// TIA Portal project "Trapano" (V15.1)

(* hardware
DEVICE "S7-1200 station_1"  S7-1200 Station
   slot 0: "Telaio di montaggio_0"  S7-1200 Rack  Rack  V1.0
   slot 1: "PLC_1"  CPU 1214C DC/DC/DC  6ES7 214-1AG40-0XB0  V4.2
*)

// ===== PLC "PLC_1"  CPU 1214C DC/DC/DC =====

VAR_GLOBAL   // PLC tag table "Tabella delle variabili standard"
   "y" AT %I0.0 : Bool;
   "x" AT %I0.1 : Bool;
   "a" AT %I0.2 : Bool;
   "b" AT %I0.3 : Bool;
   "start" AT %I0.4 : Bool;
   "m" AT %I0.5 : Bool;
   "down" AT %Q0.0 : Bool;
   "up" AT %Q0.1 : Bool;
   "rotate" AT %Q0.2 : Bool;
   "oil" AT %Q0.3 : Bool;
END_VAR

VAR_GLOBAL CONSTANT   // PLC tag table "Tabella delle variabili standard"
   "tempo_raffreddamento" : Time := T#5s;
END_VAR

DATA_BLOCK "variabili_stato"   // DB1
{ S7_Optimized_Access := 'TRUE' }
VERSION : 0.1
   VAR RETAIN
      home : Bool := true;
      scendi : Bool;
      pezzo_alto : Bool;
      pezzo_alto_risalita : Bool;
      lubrifica : Bool;
      foro : Bool;
      sali : Bool;
      wait : Bool;
   END_VAR
BEGIN
END_DATA_BLOCK

// folder: System blocks/Program resources

DATA_BLOCK "IEC_Timer_0_DB"   // DB2
{ S7_Optimized_Access := 'TRUE' }
AUTHOR : Simatic
FAMILY : IEC
NAME : IEC_TMR
VERSION : 1.0
// stored: InstanceOfName IEC_TIMER
"IEC_TIMER"
BEGIN
END_DATA_BLOCK

// folder: (top level)

ORGANIZATION_BLOCK "Main"   // OB1, LAD, ProgramCycle
TITLE = "Main Program Sweep (Cycle)"
{ S7_Optimized_Access := 'TRUE' }
VERSION : 0.1
   VAR_INPUT
      Initial_Call : Bool;   // Initial call of this OB
      Remanence : Bool;   // =True, if remanent data are available
   END_VAR
   VAR_TEMP   // added for the SCL form of the ladder/FBD networks
      _w1 : Bool;
   END_VAR
BEGIN

REGION Network 1
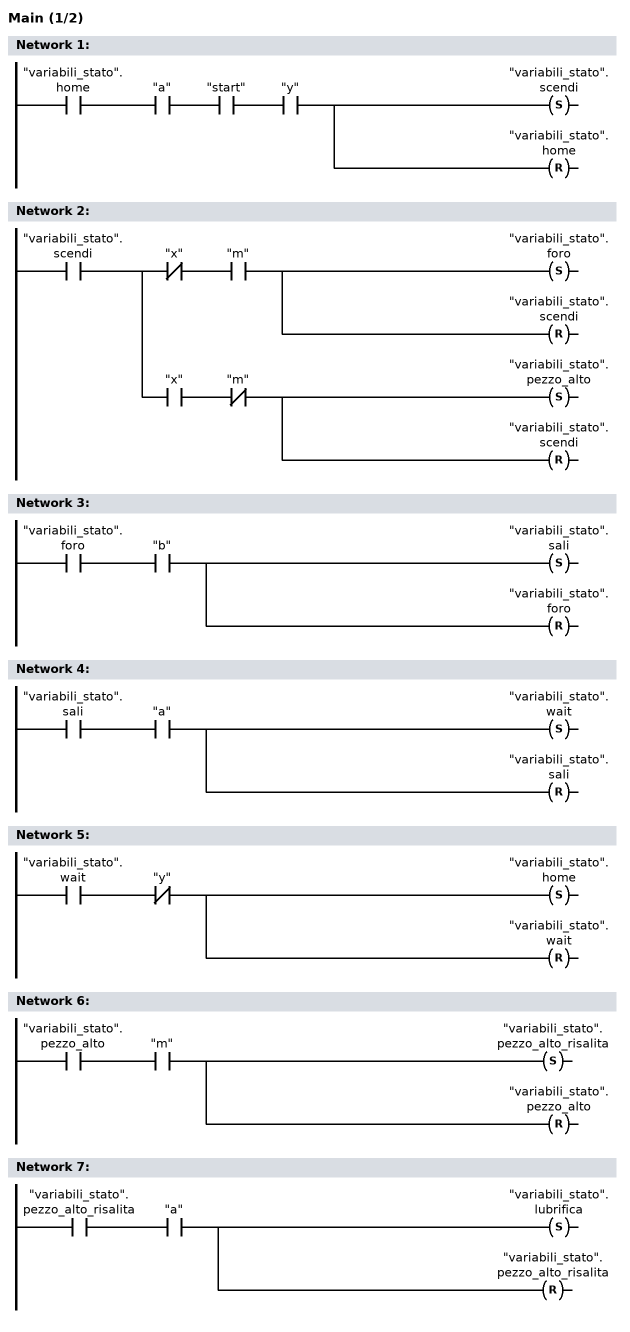
   RUNG wire#powerrail
      Contact( "variabili_stato".home )
      Contact( "a" )
      Contact( "start" )
      Contact( "y" )
      wire#w1
      S_Coil( "variabili_stato".scendi )
   END_RUNG
   RUNG wire#w1
      R_Coil( "variabili_stato".home )
   END_RUNG
   // the same network as SCL:
   IF "variabili_stato".home AND "a" AND "start" AND "y" THEN
       "variabili_stato".scendi := TRUE;
       "variabili_stato".home := FALSE;
   END_IF;
END_REGION

REGION Network 2
   RUNG wire#powerrail
      Contact( "variabili_stato".scendi )
      wire#w1
      I_Contact( "x" )
      Contact( "m" )
      wire#w2
      S_Coil( "variabili_stato".foro )
   END_RUNG
   RUNG wire#w2
      R_Coil( "variabili_stato".scendi )
   END_RUNG
   RUNG wire#w1
      Contact( "x" )
      I_Contact( "m" )
      wire#w3
      S_Coil( "variabili_stato".pezzo_alto )
   END_RUNG
   RUNG wire#w3
      R_Coil( "variabili_stato".scendi )
   END_RUNG
   // the same network as SCL:
   IF "variabili_stato".scendi AND NOT "x" AND "m" THEN "variabili_stato".foro := TRUE; END_IF;
   #_w1 := "variabili_stato".scendi;
   IF "variabili_stato".scendi AND NOT "x" AND "m" THEN "variabili_stato".scendi := FALSE; END_IF;
   IF #_w1 AND "x" AND NOT "m" THEN
       "variabili_stato".pezzo_alto := TRUE;
       "variabili_stato".scendi := FALSE;
   END_IF;
END_REGION

REGION Network 3
   RUNG wire#powerrail
      Contact( "variabili_stato".foro )
      Contact( "b" )
      wire#w1
      S_Coil( "variabili_stato".sali )
   END_RUNG
   RUNG wire#w1
      R_Coil( "variabili_stato".foro )
   END_RUNG
   // the same network as SCL:
   IF "variabili_stato".foro AND "b" THEN
       "variabili_stato".sali := TRUE;
       "variabili_stato".foro := FALSE;
   END_IF;
END_REGION

REGION Network 4
   RUNG wire#powerrail
      Contact( "variabili_stato".sali )
      Contact( "a" )
      wire#w1
      S_Coil( "variabili_stato".wait )
   END_RUNG
   RUNG wire#w1
      R_Coil( "variabili_stato".sali )
   END_RUNG
   // the same network as SCL:
   IF "variabili_stato".sali AND "a" THEN
       "variabili_stato".wait := TRUE;
       "variabili_stato".sali := FALSE;
   END_IF;
END_REGION

REGION Network 5
   RUNG wire#powerrail
      Contact( "variabili_stato".wait )
      I_Contact( "y" )
      wire#w1
      S_Coil( "variabili_stato".home )
   END_RUNG
   RUNG wire#w1
      R_Coil( "variabili_stato".wait )
   END_RUNG
   // the same network as SCL:
   IF "variabili_stato".wait AND NOT "y" THEN
       "variabili_stato".home := TRUE;
       "variabili_stato".wait := FALSE;
   END_IF;
END_REGION

REGION Network 6
   RUNG wire#powerrail
      Contact( "variabili_stato".pezzo_alto )
      Contact( "m" )
      wire#w1
      S_Coil( "variabili_stato".pezzo_alto_risalita )
   END_RUNG
   RUNG wire#w1
      R_Coil( "variabili_stato".pezzo_alto )
   END_RUNG
   // the same network as SCL:
   IF "variabili_stato".pezzo_alto AND "m" THEN
       "variabili_stato".pezzo_alto_risalita := TRUE;
       "variabili_stato".pezzo_alto := FALSE;
   END_IF;
END_REGION

REGION Network 7
   RUNG wire#powerrail
      Contact( "variabili_stato".pezzo_alto_risalita )
      Contact( "a" )
      wire#w1
      S_Coil( "variabili_stato".lubrifica )
   END_RUNG
   RUNG wire#w1
      R_Coil( "variabili_stato".pezzo_alto_risalita )
   END_RUNG
   // the same network as SCL:
   IF "variabili_stato".pezzo_alto_risalita AND "a" THEN
       "variabili_stato".lubrifica := TRUE;
       "variabili_stato".pezzo_alto_risalita := FALSE;
   END_IF;
END_REGION

REGION Network 8
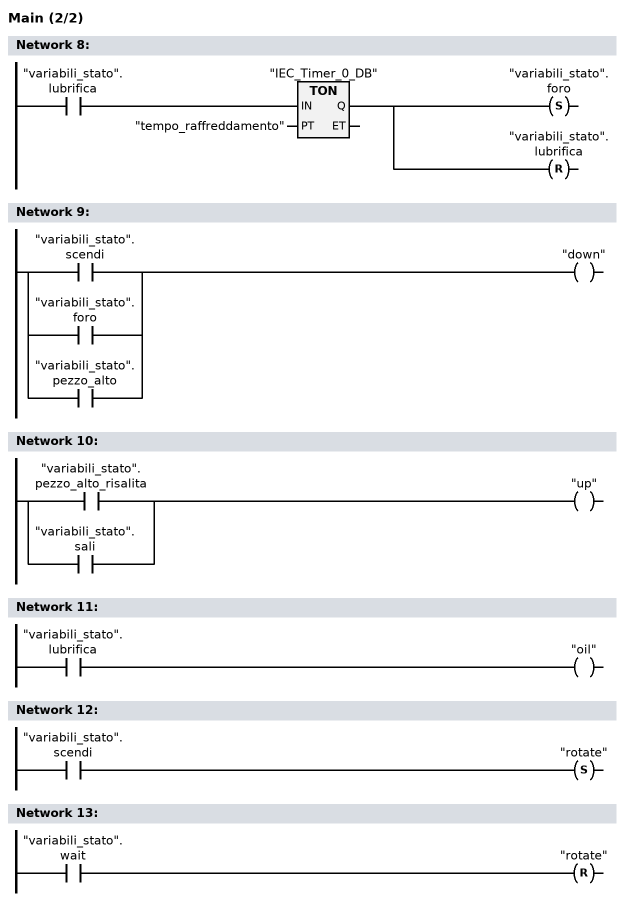
   "IEC_Timer_0_DB".TON(IN := "variabili_stato".lubrifica, PT := "tempo_raffreddamento");
   IF "IEC_Timer_0_DB".Q THEN
       "variabili_stato".foro := TRUE;
       "variabili_stato".lubrifica := FALSE;
   END_IF;
END_REGION

REGION Network 9
   RUNG wire#powerrail
      Contact( "variabili_stato".scendi )
      wire#w1
      Coil( "down" )
   END_RUNG
   RUNG wire#powerrail
      Contact( "variabili_stato".foro )
   END_RUNG wire#w1
   RUNG wire#powerrail
      Contact( "variabili_stato".pezzo_alto )
   END_RUNG wire#w1
   // the same network as SCL:
   "down" := "variabili_stato".scendi OR "variabili_stato".foro OR "variabili_stato".pezzo_alto;
END_REGION

REGION Network 10
   RUNG wire#powerrail
      Contact( "variabili_stato".pezzo_alto_risalita )
      wire#w1
      Coil( "up" )
   END_RUNG
   RUNG wire#powerrail
      Contact( "variabili_stato".sali )
   END_RUNG wire#w1
   // the same network as SCL:
   "up" := "variabili_stato".pezzo_alto_risalita OR "variabili_stato".sali;
END_REGION

REGION Network 11
   RUNG wire#powerrail
      Contact( "variabili_stato".lubrifica )
      Coil( "oil" )
   END_RUNG
   // the same network as SCL:
   "oil" := "variabili_stato".lubrifica;
END_REGION

REGION Network 12
   RUNG wire#powerrail
      Contact( "variabili_stato".scendi )
      S_Coil( "rotate" )
   END_RUNG
   // the same network as SCL:
   IF "variabili_stato".scendi THEN "rotate" := TRUE; END_IF;
END_REGION

REGION Network 13
   RUNG wire#powerrail
      Contact( "variabili_stato".wait )
      R_Coil( "rotate" )
   END_RUNG
   // the same network as SCL:
   IF "variabili_stato".wait THEN "rotate" := FALSE; END_IF;
END_REGION
END_ORGANIZATION_BLOCK